(* PLC project FBInterlockDemo, DemoCo plc-emu 0.1.0 *)
(* stored: creationDateTime 2025-11-20T00:00:00Z, modificationDateTime 2025-11-20T00:00:00Z, version 1.0, organization DemoCo *)

FUNCTION_BLOCK FB_MotorInterlock
  VAR_INPUT
    Cmd : BOOL;
    AlarmReset : BOOL;
  END_VAR
  VAR_OUTPUT
    Out : BOOL;
    Alarm : BOOL;
  END_VAR
  VAR
    StartDelayDone : BOOL;
  END_VAR

IF Alarm THEN
    Out := FALSE;
    IF AlarmReset THEN
        Alarm := FALSE;
    END_IF;
ELSIF Cmd THEN
    StartDelayDone := TRUE;
    IF StartDelayDone THEN
        Out := TRUE;
    END_IF;
ELSE
    Out := FALSE;
END_IF;
END_FUNCTION_BLOCK

PROGRAM Main_ST
  VAR
    fbMotor : FB_MotorInterlock;
  END_VAR

fbMotor.Cmd := StartPB AND NOT StopPB;
fbMotor.AlarmReset := FALSE;
fbMotor(); (* execute FB *)
MotorOut := fbMotor.Out;
Alarm := fbMotor.Alarm;
END_PROGRAM

CONFIGURATION Config0
  VAR_GLOBAL
    StartPB AT %IX0.0 : BOOL;
    StopPB AT %IX0.1 : BOOL;
    MotorOut AT %QX0.0 : BOOL;
    Alarm : BOOL;
  END_VAR
  RESOURCE Resource1 ON PLC
    TASK CyclicTask(INTERVAL := T#50ms, PRIORITY := 1);
  END_RESOURCE
END_CONFIGURATION
